(* IEC 61131-3 sources: Lasal/CPU_5344_V01/Class/checkRightOperationId1, 1 file *)

(* ---- checkRightOperationId1.st ---- *)
(*!
<Class
	Name               = "checkRightOperationId1"
	Revision           = "0.0"
	RealtimeTask       = "false"
	CyclicTask         = "false"
	BackgroundTask     = "false"
	Sigmatek           = "false"
	OSInterface        = "false"
	HighPriority       = "false"
	Automatic          = "false"
	UpdateMode         = "Prescan"
	SharedCommandTable = "true"
	Objectsize         = "(284,120)">
	<Channels>
		<Server Name="ClassSvr" Visualized="false" Initialize="false" WriteProtected="false" Retentive="false"/>
		<Server Name="maxLengthForWasteBin" Visualized="false" Initialize="true" DefValue="3000" WriteProtected="true" Retentive="false"/>
		<Server Name="minLengthForRollers" Visualized="false" Initialize="true" DefValue="5000" WriteProtected="true" Retentive="false"/>
	</Channels>
</Class>
*)
checkRightOperationId1 : CLASS
  //Servers:
	ClassSvr 	: SvrChCmd_DINT;
	minLengthForRollers 	: SvrCh_DINT;
	maxLengthForWasteBin 	: SvrCh_DINT;
  //Clients:
  //Variables:
  //Functions:

	FUNCTION GLOBAL checkMagazin
		VAR_INPUT
			iProductLength 	: DINT;
			ioOperationID1 	: DINT;
		END_VAR
		VAR_OUTPUT
			newMagazinValue 	: DINT;
		END_VAR;
  //Tables:
	FUNCTION @STD
		VAR_OUTPUT
			ret_code	: CONFSTATES;
		END_VAR;
	FUNCTION GLOBAL TAB @CT_;
END_CLASS;

FUNCTION GLOBAL checkRightOperationId1::checkMagazin
	VAR_INPUT
		iProductLength 	: DINT;
		ioOperationID1 	: DINT;
	END_VAR
	VAR_OUTPUT
		newMagazinValue 	: DINT;
	END_VAR

  newMagazinValue:=0;

  CASE ioOperationId1 OF

  1, 2, 3: //belt magazins
    IF iProductLength < maxLengthForWasteBin THEN //it fits in waste bin, so its to small for the rollers
      newMagazinValue:=10; //waste bin
    ELSIF iProductLength < minLengthForRollers THEN //to small for rollers to big for waste bin, take out manually
      newMagazinValue:=11; //take out manually
    END_IF;

  10: //waste bin
    IF iProductLength > maxLengthForWasteBin THEN //to big for waste bin
      IF iProductLength <= minLengthForRollers THEN //to small for rollers to big for waste bin, take out manually
        newMagazinValue:=11; //take out manually
      ELSE //fits in rollers
        newMagazinValue:=3; //let machine choose roller
      END_IF;
    END_IF;

  11: //always ok

  ELSE //no proper choice made

    IF iProductLength <= maxLengthForWasteBin THEN //it fits in waste bin, so its to small for the rollers
      newMagazinValue:=10; //waste bin
    ELSIF iProductLength <= minLengthForRollers THEN //to small for rollers to big for waste bin, take out manually
      newMagazinValue:=11; //take out manually
    ELSE //fits in rollers
      newMagazinValue:=3; //let machine choose roller
    END_IF;

  END_CASE;

END_FUNCTION
